FUNCTION_BLOCK SLEEP
  {SET_ATTRIBUTE(OpcUa, DEVICE.SENSOR)}
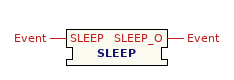
  EVENT_INPUT
    SLEEP;
  END_EVENT
  EVENT_OUTPUT
    SLEEP_O;
  END_EVENT
END_FUNCTION_BLOCK
